FUNCTION_BLOCK FAN_VOLTAGE_CONTROL EXTENDS FB_CONTROL 
VAR
	fbOutput		: FB_OutLinear;
END_VAR

METHOD Control
IF fSet < 0 THEN
	fSet := 0;
END_IF

SUPER^.Control();
END_METHOD

PROPERTY Output : REFERENCE TO FB_OutLinear
GET
Output REF=THIS^.fbOutput;
END_GET
END_PROPERTY

METHOD Write
fbOutput.ValueOut := SUPER^.fY;
IF fSet <= 0 THEN
	fbOutput.ValueOut := 0;
END_IF
fbOutput.Write();
END_METHOD

END_FUNCTION_BLOCK

(* stored: Version 1.1.0.1, ProductVersion 3.1.4024.3
   POU FAN_VOLTAGE_CONTROL: Id {46b85e44-dde3-42b1-aa18-ffc577baf9f6}, SpecialFunc None
   Method Control: Id {22213b50-62cb-46cc-9d2f-09585c7911d3}
   Property Output: Id {9a1e45b0-0f6e-4273-aa0d-7545de409a58}
   Get Get: Id {b2ea25cc-1729-432b-ae06-ce2da8038476}
   Method Write: Id {9d476219-2625-46a7-9000-7861cc0be81d} *)
